Staubli VAL3: sendPowerOff.pgx

program sendPowerOff()
  local num buffer[2]
begin
  buffer[0] = MAGIC_HEADER
  buffer[1] = 130
  sioSet(socket, buffer)
end
